# EPICS autosave request: ADmar345/iocs/mar345IOC/iocBoot/iocMAR345/auto_settings.req
file "ADBase_settings.req",       P=$(P),  R=cam1:
file "mar345_settings.req",       P=$(P),  R=cam1:
file "NDFile_settings.req",       P=$(P),  R=cam1:
file "NDPluginBase_settings.req", P=$(P),  R=image1:
file "NDStdArrays_settings.req",  P=$(P),  R=image1:
file "commonPlugin_settings.req", P=$(P)
